//---------------------------------------------------------------------------------------------------------------
//
//  HAUD 2024.10.02
//
//  - APPLICATION
//    - explicit simple example PRG for setting up GearInPosCa application
//      - works dirEctly on GVL_XTS namespace Ctrl/State structs
//      - no error handling, reset application from start
//
//  - Application controls:
//    - XtsTransport
//      - GVL_XTS.TransportCtrl
//      - GVL_XTS.TransportState
//
//    - Xts Movers
//      - GVL_XTS.MoverCtrl
//      - GVL_XTS.MoverState
//      - GVL_XTS.MoverInfo
//      - GVL_XTS.MoveData
//      - GVL_XTS.GearData
//
//  - Application
//    - GearInPosCa example
//      - gear in to conveyer belt 
//
//---------------------------------------------------------------------------------------------------------------
// This SOFTWARE is provided as an Exemple by THE PROVIDER "as is" and "with all faults." THE PROVIDER makes no 
// representations or warranties of any kind concerning the safety, suitability, lack of viruses, inaccuracies, 
// typographical errors, or other harmful components of this SOFTWARE. There are inherent dangers in the use of 
// any software, and you are solely responsible for determining whether this SOFTWARE is compatible with your 
// equipment and other software installed on your equipment. You are also solely responsible for the protection 
// of your equipment and backup of your data, and THE PROVIDER will not be liable for any damages you may suffer 
// in connection with using, modifying, or distributing this SOFTWARE.
//---------------------------------------------------------------------------------------------------------------
PROGRAM APPLICATION
VAR
  eInit         : E_PROGRESS;
  bStart        : BOOL;   // XtsTransport is initialized, CAGroup is built, All movers are enabled, XtsStations are cleared, XtsTransport base position for all movers is commanded, XtsStations are handshaked with timer
  bReset        : BOOL;   // All Xts Stations are cleared, requires new start

  nState        : UINT;   // state var for application
END_VAR



//-----------------------------------------------------------------------------
// wait for initialization to be complete before work may start
//-----------------------------------------------------------------------------
IF NOT (Main.eInit = E_PROGRESS.PROGRESS_DONE)
THEN
  eInit                               := E_PROGRESS.PROGRESS_INIT;
  bReset                              := FALSE;
  bStart                              := FALSE;
  nState                              := 0;
  RETURN;
END_IF
//-----------------------------------------------------------------------------
// fetch reset anytime
//-----------------------------------------------------------------------------
IF bReset
THEN
  bReset                              := FALSE;
  bStart                              := FALSE;
  nState                              := 9000;  // states for clearing XtsTransport
END_IF


CASE nState 
OF
  0:                                  // first PLC cycle
    nState                            := 1;

  1:
    // do other init stuff here
    eInit                             := E_PROGRESS.PROGRESS_DONE;
    nState                            := 10;

  10:                                 // starts from here
    IF bStart
    THEN
      nState                          := 100; // let's go
    END_IF
    
  100:                                // clear interface
    GVL_XTS.XtsTransportCtrl.Cmd      := E_XTS_TRANSPORT_CTRL.CMD_NULL;
    nState                            := 110;

  110:                                // check initialization of XtsTransport, wait for either MoverDetection being valid or OperationMode.Simulation
    IF (GVL_XTS.XtsTransportState.XpuInfo.IdDetectionValid) OR
       (GVL_XTS.XtsTransportState.XpuInfo.OperationMode = OperationMode.Simulation)
    THEN
      // now XtsTransport is initialized, cyclic plausibility checks on Xpu are active
      nState                          := 120;
    END_IF

  120:                                // clear group for defined start situation
    GVL_XTS.XtsTransportCtrl.Cmd      := E_XTS_TRANSPORT_CTRL.CMD_GROUP_CLEAR;

    IF (GVL_XTS.XtsTransportState.State = E_XTS_TRANSPORT_STATE.TRANSPORT_GROUP_CLEAR + E_PROGRESS.PROGRESS_DONE)
    THEN
      // CA Group is now in defined error free state
      nState                          := 130;
    END_IF

  130:                                // build Collision Avoidance group with all movers
    GVL_XTS.XtsTransportCtrl.Cmd      := E_XTS_TRANSPORT_CTRL.CMD_GROUP_BUILD;

    IF (GVL_XTS.XtsTransportState.State = E_XTS_TRANSPORT_STATE.TRANSPORT_GROUP_BUILD + E_PROGRESS.PROGRESS_DONE)
    THEN
      // CA Group contains all movers now
      // GVL_XTS.XtsTransportState.GroupInfo.AxisCount = MAX_MOVER
      nState                          := 140;
      GEAR_IN_POS_CA.bEnable          := FALSE;
      GEAR_IN_POS_CA.bReset           := FALSE;
    END_IF

  140:                                // enable CA Group
    GVL_XTS.XtsTransportCtrl.Cmd      := E_XTS_TRANSPORT_CTRL.CMD_GROUP_ENABLE;

    IF (GVL_XTS.XtsTransportState.State = E_XTS_TRANSPORT_STATE.TRANSPORT_GROUP_ENABLE + E_PROGRESS.PROGRESS_DONE)
    THEN
      // GVL_XTS.XtsTransportState.GroupInfo.CaGroupState = mcGroupStateNotReady
      nState                          := 150;
      GEAR_IN_POS_CA.bReset           := TRUE;
    END_IF

  150:                                // enable all movers
    GVL_XTS.XtsTransportCtrl.Cmd      := E_XTS_TRANSPORT_CTRL.CMD_MOVER_ENABLE;

    IF (GVL_XTS.XtsTransportState.State = E_XTS_TRANSPORT_STATE.TRANSPORT_MOVER_ENABLE + E_PROGRESS.PROGRESS_DONE)
    THEN
      // GVL_XTS.XtsTransportState.GroupInfo.CaGroupState = mcGroupStateStandby
      nState                          := 160;
      GEAR_IN_POS_CA.bReset           := FALSE;
    END_IF

  160:                                // command all movers to startup position
    GVL_XTS.XtsTransportCtrl.Cmd      := E_XTS_TRANSPORT_CTRL.CMD_TRANSPORT_START;

    IF (GVL_XTS.XtsTransportState.State = E_XTS_TRANSPORT_STATE.TRANSPORT_START + E_PROGRESS.PROGRESS_DONE)
    THEN
      // all movers are now waiting at GVL_XTS.StationStart.rPosWait
      nState                          := 1000; // go to wait state, activate GearInPos program
      // enable gear in pos sequence now the movers are ready
      GEAR_IN_POS_CA.bEnable          := TRUE;
    END_IF


  9000:
    // reset sequence trigger starts here
    GEAR_IN_POS_CA.bEnable            := FALSE;
    GVL_XTS.XtsTransportCtrl.Cmd      := E_XTS_TRANSPORT_CTRL.CMD_NULL;
    nState                            := 9005;

    GVL_APPLICATION.MasterHalt(
                        Axis          := GVL_APPLICATION.MasterAxis, 
                        Execute       := FALSE, 
                        Deceleration  :=  12500.0, 
                        Jerk          := 100000.0, 
                        BufferMode    := Tc2_MC2.MC_Aborting, 
                        Options:= , 
                        Done=> , 
                        Busy=> , 
                        Active=> , 
                        CommandAborted=> , 
                        Error=> , 
                        ErrorID=> );

  9005:
    GVL_APPLICATION.MasterHalt(
                        Axis          := GVL_APPLICATION.MasterAxis, 
                        Execute       := TRUE);

    IF (GVL_APPLICATION.MasterAxis.Status.NotMoving)
    THEN
      nState                          := 9010;

      GVL_APPLICATION.MasterHalt(
                          Axis        := GVL_APPLICATION.MasterAxis, 
                          Execute     := FALSE);

      GVL_APPLICATION.MasterPower(
                  Axis                := GVL_APPLICATION.MasterAxis, 
                  Enable              := FALSE);
    END_IF

  9010:                               // halt all movers and clear group
    GVL_XTS.XtsTransportCtrl.Cmd      := E_XTS_TRANSPORT_CTRL.CMD_GROUP_CLEAR;

    IF (GVL_XTS.XtsTransportState.State = E_XTS_TRANSPORT_STATE.TRANSPORT_GROUP_CLEAR + E_PROGRESS.PROGRESS_DONE)
    THEN
      // CA group cleared and mover in standstill
      nState                          := 9100;
    END_IF

  9100:                               // switch off movers
    GVL_XTS.XtsTransportCtrl.Cmd      := E_XTS_TRANSPORT_CTRL.CMD_MOVER_DISABLE;

    IF (GVL_XTS.XtsTransportState.State = E_XTS_TRANSPORT_STATE.TRANSPORT_MOVER_DISABLE + E_PROGRESS.PROGRESS_ERROR)
    THEN
      nState                          := 9010;
    ELSIF (GVL_XTS.XtsTransportState.State = E_XTS_TRANSPORT_STATE.TRANSPORT_MOVER_DISABLE + E_PROGRESS.PROGRESS_DONE)
    THEN
      nState                          := 10;
    END_IF

END_CASE

GVL_APPLICATION.MasterAxis(); // update master axis

GEAR_IN_POS_CA();             // gear in pos sequence

END_PROGRAM

(* stored: Version 1.1.0.1, ProductVersion 3.1.4024.13
   POU APPLICATION: Id {a42cfa77-97a5-4ec9-b576-fd1e63c4d66c}, SpecialFunc None *)
